Staubli VAL3: frmtool.pjx

--- frmtool.pjx ---
Parameters version=s7.8.2 stackSize=5000 millimeterUnit=true
Program file=start.pgx
Program file=stop.pgx
Data file=frmtool.dtx

--- frmtool.dtx ---
mdesc mNomSpeed
public frame frmaster = {fatherId=world[0]}
public tool t2[10]
  [0] = {fatherId=flange[0], ioLink=valve1}
  [1] = {fatherId=flange[0], ioLink=valve1}
  [2] = {fatherId=flange[0], ioLink=valve1}
  [3] = {fatherId=flange[0], ioLink=valve1}
  [4] = {fatherId=flange[0], ioLink=valve1}
  [5] = {fatherId=flange[0], ioLink=valve1}
  [6] = {fatherId=flange[0], ioLink=valve1}
  [7] = {fatherId=flange[0], ioLink=valve1}
  [8] = {fatherId=flange[0], ioLink=valve1}
  [9] = {fatherId=flange[0], ioLink=valve1}
public tool t1 = {fatherId=flange[0], ioLink=valve1}
public frame fr1 = {fatherId=world[0]}
